SUBAPPLICATION Q_BackgroundColour_EnableOk_AX (* Wie MyLib::sys::Q_BackgroundColour_EnableOk, aber bEnable/bOk kommen als AX-Adapter (statt Klartext-BOOL) - Stil/Schnittstelle wie GreenBlueBackground1_AX (nur CNF, kein REQ; STATUS_1/u8OldColour_1/result_1). *)
  (* Standard: 61499-2; Description: Copyright (c) 2026 Meisterschulen am Ostbahnhof This program and the accompanying materials are made available under the terms of the Eclipse Public License 2.0 which is available at https://www.eclipse.org/legal/epl-2.0/ SPDX-License-Identifier: EPL-2.0 *)
  (* Version 1.0, 2026-08-31, Franz Höpfinger, Meisterschulen am Ostbahnhof, AX-Adapter-Variante von Q_BackgroundColour_EnableOk, im Stil der bestehenden GreenBlueBackground1_AX/GreenRedBackground1_AX-Familie *)
  PACKAGE MyLib::sys;
  IMPORT isobus::UT::Q::const::IDs::ID_NULL;
  IMPORT isobus::UT::Q::const::colours::COLOR_GREEN;
  IMPORT isobus::UT::Q::const::colours::COLOR_RED;
  IMPORT isobus::UT::Q::const::colours::COLOR_WHITE;
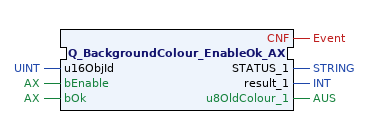
  EVENT_OUTPUT
    CNF; (* Execution Confirmation *)
  END_EVENT
  VAR_INPUT
    u16ObjId : UINT := ID_NULL; (* Object ID Status-Anzeige (CButton, nur Hintergrundfarbe, kein Text) *)
  END_VAR
  VAR_OUTPUT
    STATUS_1 : STRING; (* Service Status *)
    result_1 : INT; (* retval see description *)
  END_VAR
  SOCKETS
    bEnable : adapter::types::unidirectional::AX; (* Aktiviert (BOOL, ueber Adapter statt Klartext) *)
    bOk : adapter::types::unidirectional::AX; (* OK-Zustand (BOOL, ueber Adapter statt Klartext) - nur relevant wenn bEnable=TRUE *)
  END_SOCKETS
  PLUGS
    u8OldColour_1 : adapter::types::unidirectional::AUS; (* Old value of ID *)
  END_PLUGS
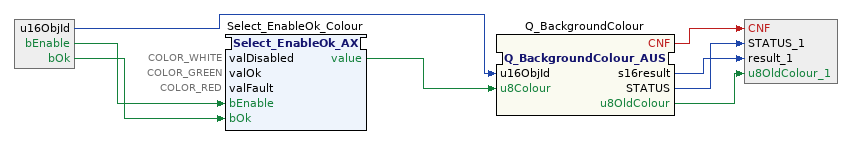
  FBS
    Q_BackgroundColour : isobus::UT::Q::Q_BackgroundColour_AUS;
  END_FBS
  SUBAPPS
    Select_EnableOk_Colour : MyLib::sys::Select_EnableOk_AX(valDisabled := COLOR_WHITE, valOk := COLOR_GREEN, valFault := COLOR_RED);
  END_SUBAPPS
  EVENT_CONNECTIONS
    Q_BackgroundColour.CNF TO CNF;
  END_CONNECTIONS
  DATA_CONNECTIONS
    u16ObjId TO Q_BackgroundColour.u16ObjId;
    Q_BackgroundColour.s16result TO result_1;
    Q_BackgroundColour.STATUS TO STATUS_1;
  END_CONNECTIONS
  ADAPTER_CONNECTIONS
    bEnable TO Select_EnableOk_Colour.bEnable;
    bOk TO Select_EnableOk_Colour.bOk;
    Select_EnableOk_Colour.value TO Q_BackgroundColour.u8Colour;
    Q_BackgroundColour.u8OldColour TO u8OldColour_1;
  END_CONNECTIONS
END_SUBAPPLICATION
